// Mitsubishi GX Works2 project: elevator-finished-fixed   PLC: FX3U/FX3UC

PROGRAM MAIN
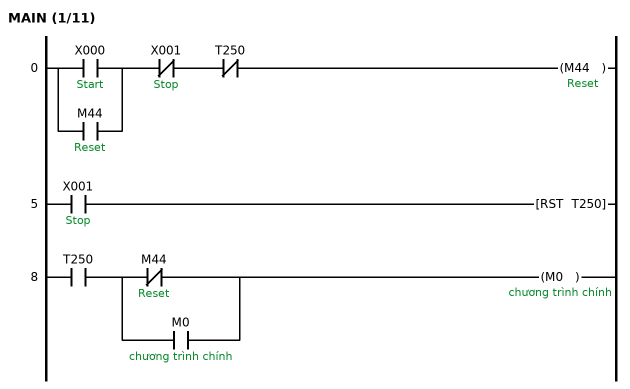
0     LD      X000  ; Start
      OR      M44  ; Reset
      ANI     X001  ; Stop
      ANI     T250
      OUT     M44  ; Reset
5     LD      X001  ; Stop
      RST     T250
8     LD      T250
      LDI     M44  ; Reset
      OR      M0  ; chương trình chính
      ANB
      OUT     M0  ; chương trình chính
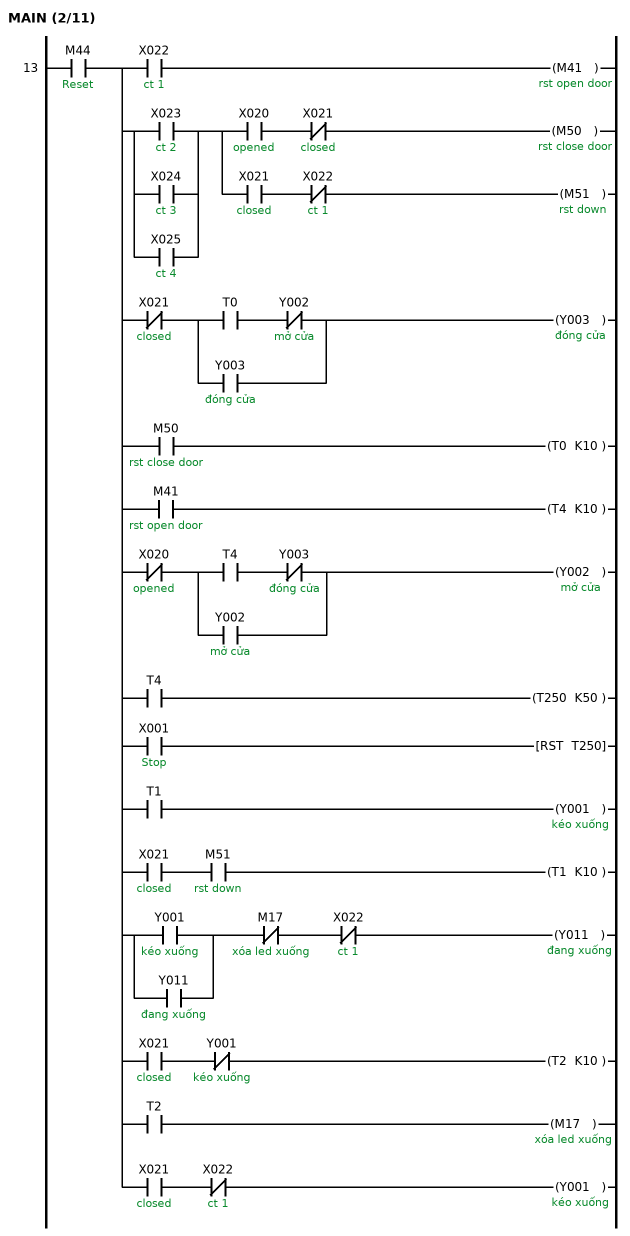
13    LD      M44  ; Reset
      MPS
      AND     X022  ; ct 1
      OUT     M41  ; rst open door
      MRD
      LD      X023  ; ct 2
      OR      X024  ; ct 3
      OR      X025  ; ct 4
      ANB
      MPS
      AND     X020  ; opened
      ANI     X021  ; closed
      OUT     M50  ; rst close door
      MPP
      AND     X021  ; closed
      ANI     X022  ; ct 1
      OUT     M51  ; rst down
      MRD
      ANI     X021  ; closed
      LD      T0
      ANI     Y002  ; mở cửa
      OR      Y003  ; đóng cửa
      ANB
      OUT     Y003  ; đóng cửa
      MRD
      AND     M50  ; rst close door
      OUT     T0 K10
      MRD
      AND     M41  ; rst open door
      OUT     T4 K10
      MRD
      ANI     X020  ; opened
      LD      T4
      ANI     Y003  ; đóng cửa
      OR      Y002  ; mở cửa
      ANB
      OUT     Y002  ; mở cửa
      MRD
      AND     T4
      OUT     T250 K50
      MRD
      AND     X001  ; Stop
      RST     T250
      MRD
      AND     T1
      OUT     Y001  ; kéo xuống
      MRD
      AND     X021  ; closed
      AND     M51  ; rst down
      OUT     T1 K10
      MRD
      LD      Y001  ; kéo xuống
      OR      Y011  ; đang xuống
      ANB
      ANI     M17  ; xóa led xuống
      ANI     X022  ; ct 1
      OUT     Y011  ; đang xuống
      MRD
      AND     X021  ; closed
      ANI     Y001  ; kéo xuống
      OUT     T2 K10
      MRD
      AND     T2
      OUT     M17  ; xóa led xuống
      MPP
      AND     X021  ; closed
      ANI     X022  ; ct 1
      OUT     Y001  ; kéo xuống
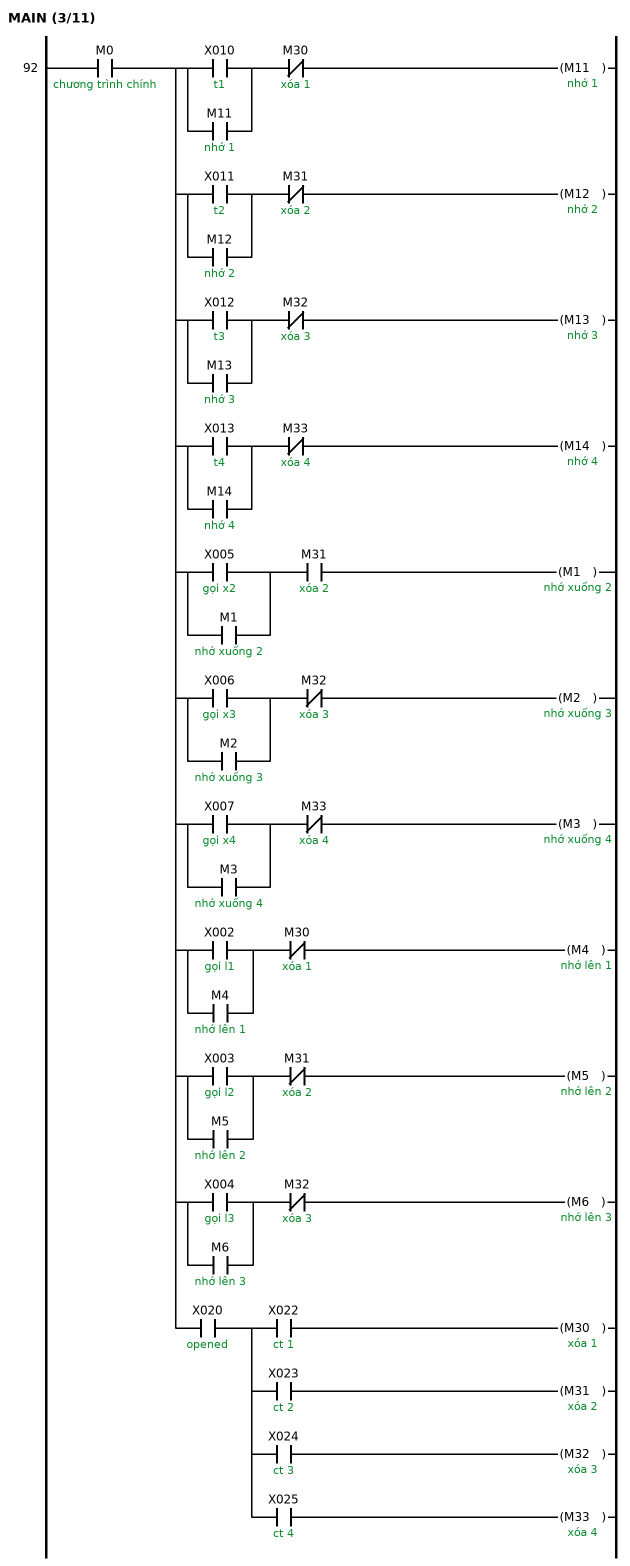
92    LD      M0  ; chương trình chính
      MPS
      LD      X010  ; t1
      OR      M11  ; nhớ 1
      ANB
      ANI     M30  ; xóa 1
      OUT     M11  ; nhớ 1
      MRD
      LD      X011  ; t2
      OR      M12  ; nhớ 2
      ANB
      ANI     M31  ; xóa 2
      OUT     M12  ; nhớ 2
      MRD
      LD      X012  ; t3
      OR      M13  ; nhớ 3
      ANB
      ANI     M32  ; xóa 3
      OUT     M13  ; nhớ 3
      MRD
      LD      X013  ; t4
      OR      M14  ; nhớ 4
      ANB
      ANI     M33  ; xóa 4
      OUT     M14  ; nhớ 4
      MRD
      LD      X005  ; gọi x2
      OR      M1  ; nhớ xuống 2
      ANB
      AND     M31  ; xóa 2
      OUT     M1  ; nhớ xuống 2
      MRD
      LD      X006  ; gọi x3
      OR      M2  ; nhớ xuống 3
      ANB
      ANI     M32  ; xóa 3
      OUT     M2  ; nhớ xuống 3
      MRD
      LD      X007  ; gọi x4
      OR      M3  ; nhớ xuống 4
      ANB
      ANI     M33  ; xóa 4
      OUT     M3  ; nhớ xuống 4
      MRD
      LD      X002  ; gọi l1
      OR      M4  ; nhớ lên 1
      ANB
      ANI     M30  ; xóa 1
      OUT     M4  ; nhớ lên 1
      MRD
      LD      X003  ; gọi l2
      OR      M5  ; nhớ lên 2
      ANB
      ANI     M31  ; xóa 2
      OUT     M5  ; nhớ lên 2
      MRD
      LD      X004  ; gọi l3
      OR      M6  ; nhớ lên 3
      ANB
      ANI     M32  ; xóa 3
      OUT     M6  ; nhớ lên 3
      MPP
      AND     X020  ; opened
      MPS
      AND     X022  ; ct 1
      OUT     M30  ; xóa 1
      MRD
      AND     X023  ; ct 2
      OUT     M31  ; xóa 2
      MRD
      AND     X024  ; ct 3
      OUT     M32  ; xóa 3
      MPP
      AND     X025  ; ct 4
      OUT     M33  ; xóa 4
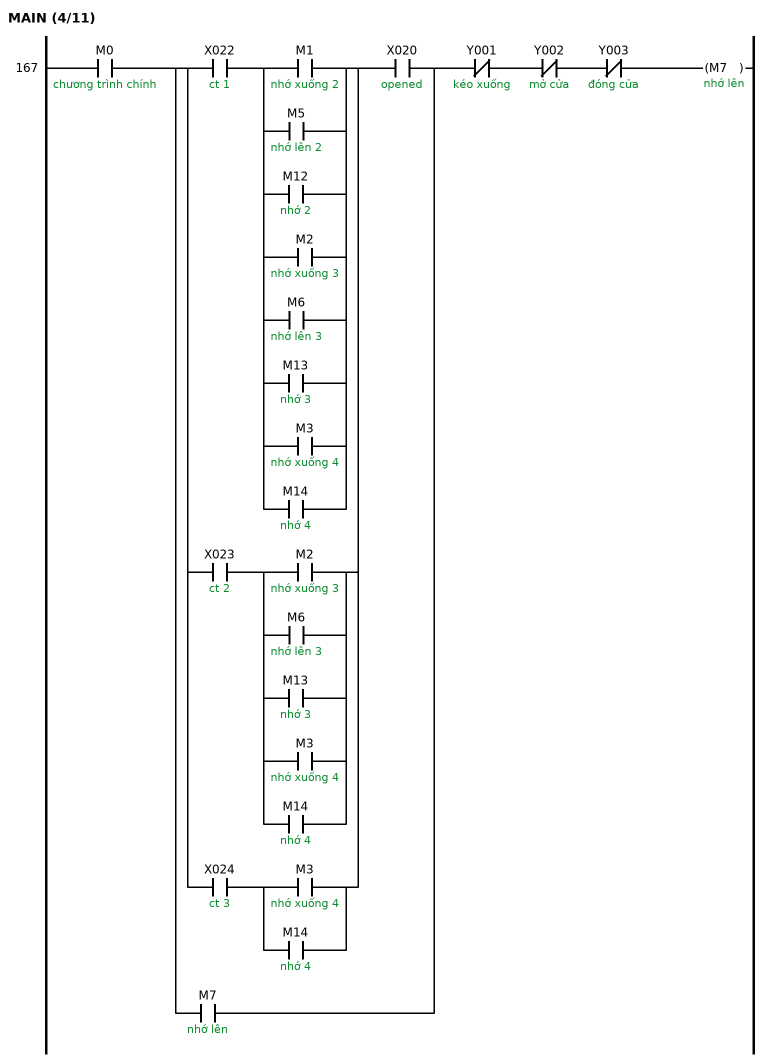
167   LD      M0  ; chương trình chính
      LD      X022  ; ct 1
      LD      M1  ; nhớ xuống 2
      OR      M5  ; nhớ lên 2
      OR      M12  ; nhớ 2
      OR      M2  ; nhớ xuống 3
      OR      M6  ; nhớ lên 3
      OR      M13  ; nhớ 3
      OR      M3  ; nhớ xuống 4
      OR      M14  ; nhớ 4
      ANB
      LD      X023  ; ct 2
      LD      M2  ; nhớ xuống 3
      OR      M6  ; nhớ lên 3
      OR      M13  ; nhớ 3
      OR      M3  ; nhớ xuống 4
      OR      M14  ; nhớ 4
      ANB
      ORB
      LD      X024  ; ct 3
      LD      M3  ; nhớ xuống 4
      OR      M14  ; nhớ 4
      ANB
      ORB
      AND     X020  ; opened
      OR      M7  ; nhớ lên
      ANB
      ANI     Y001  ; kéo xuống
      ANI     Y002  ; mở cửa
      ANI     Y003  ; đóng cửa
      OUT     M7  ; nhớ lên
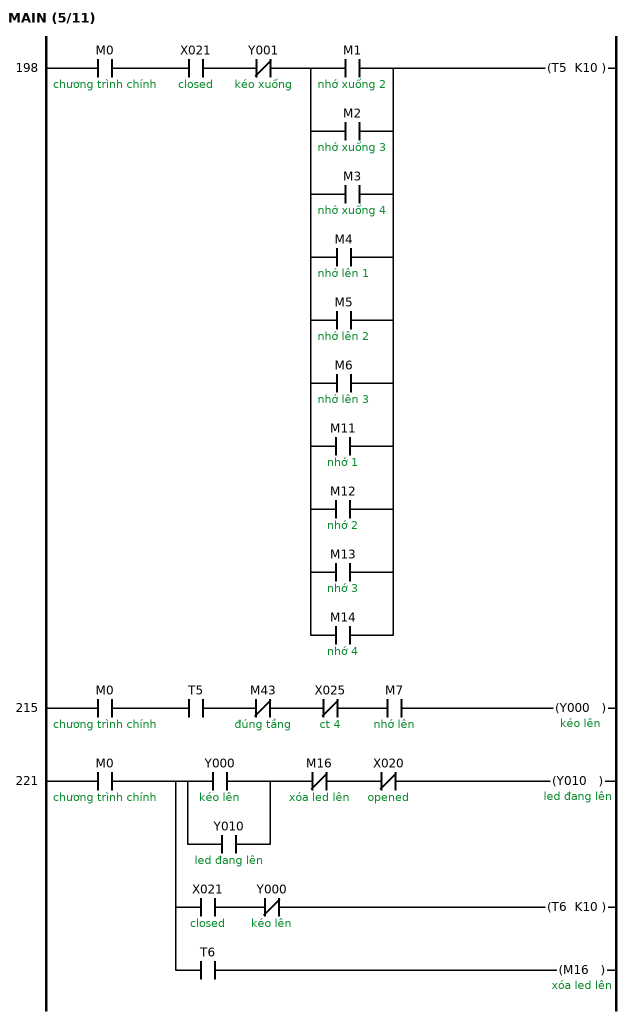
198   LD      M0  ; chương trình chính
      AND     X021  ; closed
      ANI     Y001  ; kéo xuống
      LD      M1  ; nhớ xuống 2
      OR      M2  ; nhớ xuống 3
      OR      M3  ; nhớ xuống 4
      OR      M4  ; nhớ lên 1
      OR      M5  ; nhớ lên 2
      OR      M6  ; nhớ lên 3
      OR      M11  ; nhớ 1
      OR      M12  ; nhớ 2
      OR      M13  ; nhớ 3
      OR      M14  ; nhớ 4
      ANB
      OUT     T5 K10
215   LD      M0  ; chương trình chính
      AND     T5
      ANI     M43  ; đúng tầng
      ANI     X025  ; ct 4
      AND     M7  ; nhớ lên
      OUT     Y000  ; kéo lên
221   LD      M0  ; chương trình chính
      MPS
      LD      Y000  ; kéo lên
      OR      Y010  ; led đang lên
      ANB
      ANI     M16  ; xóa led lên
      ANI     X020  ; opened
      OUT     Y010  ; led đang lên
      MRD
      AND     X021  ; closed
      ANI     Y000  ; kéo lên
      OUT     T6 K10
      MPP
      AND     T6
      OUT     M16  ; xóa led lên
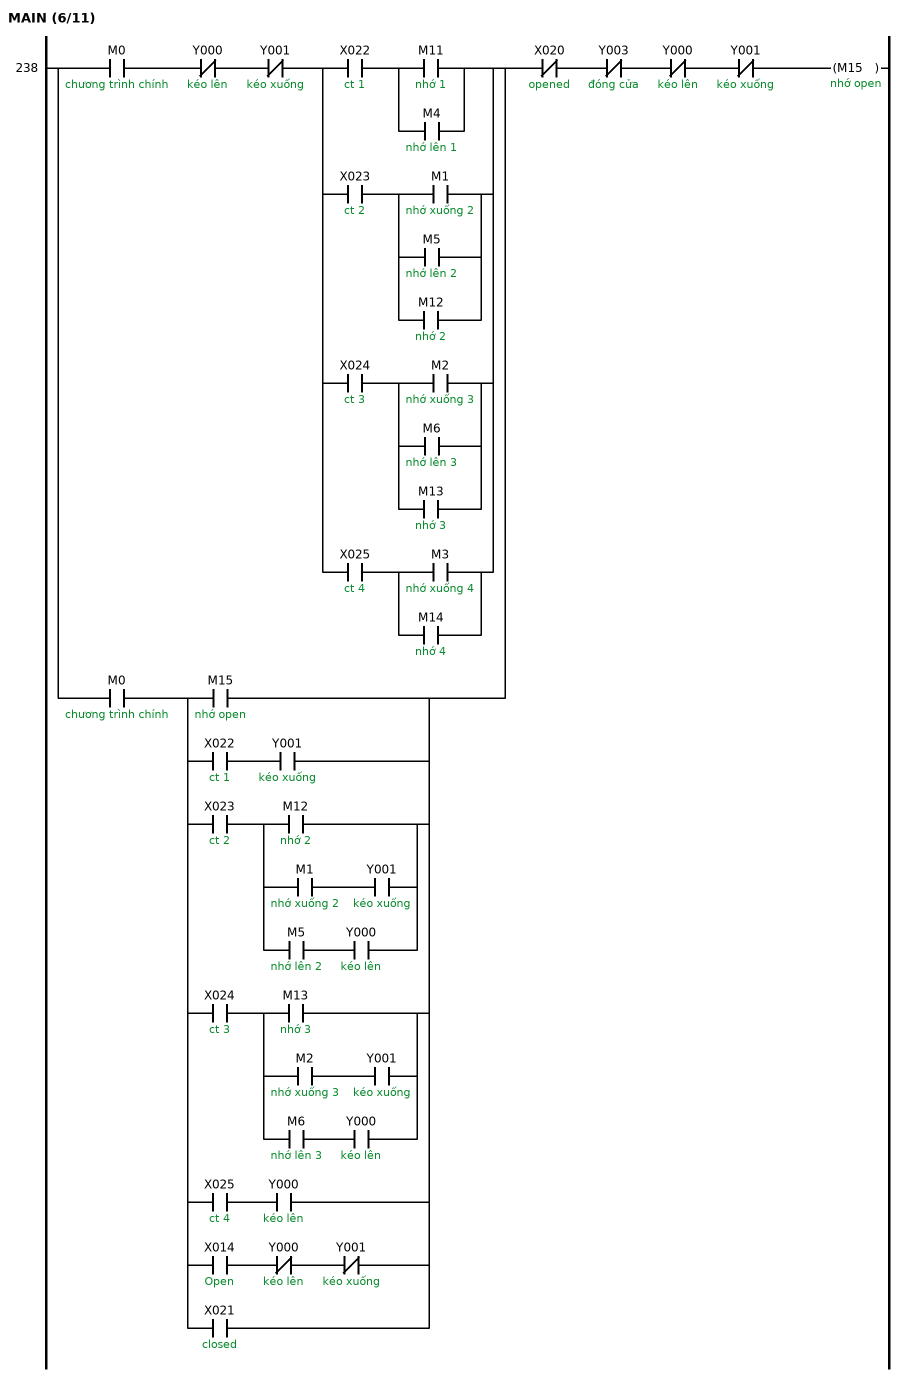
238   LD      M0  ; chương trình chính
      ANI     Y000  ; kéo lên
      ANI     Y001  ; kéo xuống
      LD      X022  ; ct 1
      LD      M11  ; nhớ 1
      OR      M4  ; nhớ lên 1
      ANB
      LD      X023  ; ct 2
      LD      M1  ; nhớ xuống 2
      OR      M5  ; nhớ lên 2
      OR      M12  ; nhớ 2
      ANB
      ORB
      LD      X024  ; ct 3
      LD      M2  ; nhớ xuống 3
      OR      M6  ; nhớ lên 3
      OR      M13  ; nhớ 3
      ANB
      ORB
      LD      X025  ; ct 4
      LD      M3  ; nhớ xuống 4
      OR      M14  ; nhớ 4
      ANB
      ORB
      ANB
      LD      M0  ; chương trình chính
      LD      M15  ; nhớ open
      LD      X022  ; ct 1
      AND     Y001  ; kéo xuống
      ORB
      LD      X023  ; ct 2
      LD      M12  ; nhớ 2
      LD      M1  ; nhớ xuống 2
      AND     Y001  ; kéo xuống
      ORB
      LD      M5  ; nhớ lên 2
      AND     Y000  ; kéo lên
      ORB
      ANB
      ORB
      LD      X024  ; ct 3
      LD      M13  ; nhớ 3
      LD      M2  ; nhớ xuống 3
      AND     Y001  ; kéo xuống
      ORB
      LD      M6  ; nhớ lên 3
      AND     Y000  ; kéo lên
      ORB
      ANB
      ORB
      LD      X025  ; ct 4
      AND     Y000  ; kéo lên
      ORB
      LD      X014  ; Open
      ANI     Y000  ; kéo lên
      ANI     Y001  ; kéo xuống
      ORB
      OR      X021  ; closed
      ANB
      ORB
      ANI     X020  ; opened
      ANI     Y003  ; đóng cửa
      ANI     Y000  ; kéo lên
      ANI     Y001  ; kéo xuống
      OUT     M15  ; nhớ open
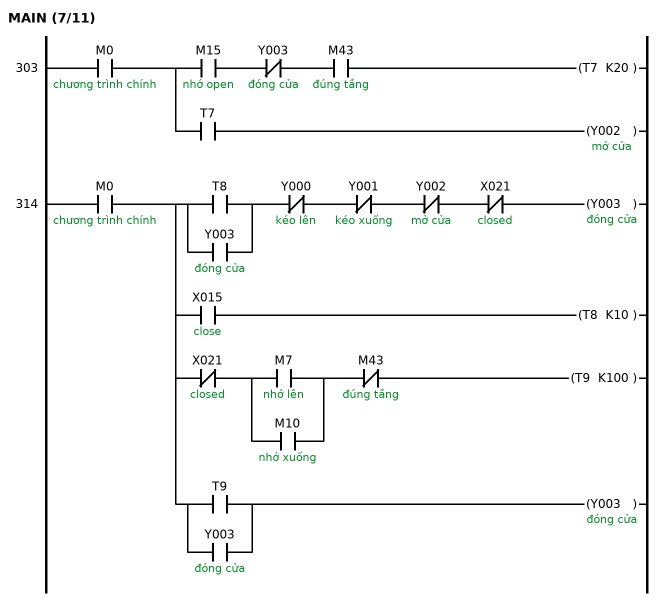
303   LD      M0  ; chương trình chính
      MPS
      AND     M15  ; nhớ open
      ANI     Y003  ; đóng cửa
      AND     M43  ; đúng tầng
      OUT     T7 K20
      MPP
      AND     T7
      OUT     Y002  ; mở cửa
314   LD      M0  ; chương trình chính
      MPS
      LD      T8
      OR      Y003  ; đóng cửa
      ANB
      ANI     Y000  ; kéo lên
      ANI     Y001  ; kéo xuống
      ANI     Y002  ; mở cửa
      ANI     X021  ; closed
      OUT     Y003  ; đóng cửa
      MRD
      AND     X015  ; close
      OUT     T8 K10
      MRD
      ANI     X021  ; closed
      LD      M7  ; nhớ lên
      OR      M10  ; nhớ xuống
      ANB
      ANI     M43  ; đúng tầng
      OUT     T9 K100
      MPP
      LD      T9
      OR      Y003  ; đóng cửa
      ANB
      OUT     Y003  ; đóng cửa
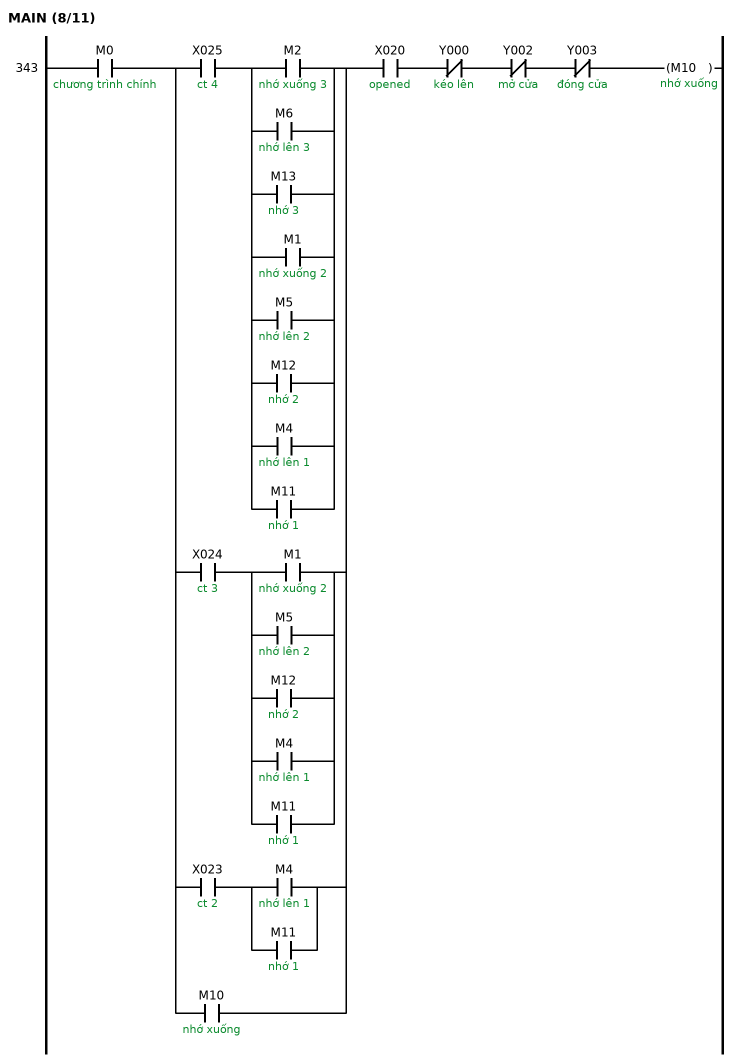
343   LD      M0  ; chương trình chính
      LD      X025  ; ct 4
      LD      M2  ; nhớ xuống 3
      OR      M6  ; nhớ lên 3
      OR      M13  ; nhớ 3
      OR      M1  ; nhớ xuống 2
      OR      M5  ; nhớ lên 2
      OR      M12  ; nhớ 2
      OR      M4  ; nhớ lên 1
      OR      M11  ; nhớ 1
      ANB
      LD      X024  ; ct 3
      LD      M1  ; nhớ xuống 2
      OR      M5  ; nhớ lên 2
      OR      M12  ; nhớ 2
      OR      M4  ; nhớ lên 1
      OR      M11  ; nhớ 1
      ANB
      ORB
      LD      X023  ; ct 2
      LD      M4  ; nhớ lên 1
      OR      M11  ; nhớ 1
      ANB
      ORB
      OR      M10  ; nhớ xuống
      ANB
      AND     X020  ; opened
      ANI     Y000  ; kéo lên
      ANI     Y002  ; mở cửa
      ANI     Y003  ; đóng cửa
      OUT     M10  ; nhớ xuống
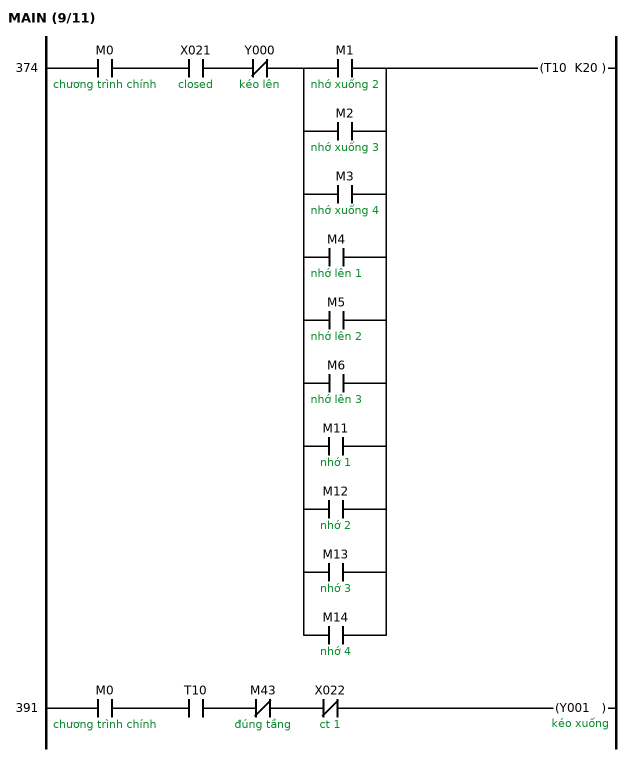
374   LD      M0  ; chương trình chính
      AND     X021  ; closed
      ANI     Y000  ; kéo lên
      LD      M1  ; nhớ xuống 2
      OR      M2  ; nhớ xuống 3
      OR      M3  ; nhớ xuống 4
      OR      M4  ; nhớ lên 1
      OR      M5  ; nhớ lên 2
      OR      M6  ; nhớ lên 3
      OR      M11  ; nhớ 1
      OR      M12  ; nhớ 2
      OR      M13  ; nhớ 3
      OR      M14  ; nhớ 4
      ANB
      OUT     T10 K20
391   LD      M0  ; chương trình chính
      AND     T10
      ANI     M43  ; đúng tầng
      ANI     X022  ; ct 1
      OUT     Y001  ; kéo xuống
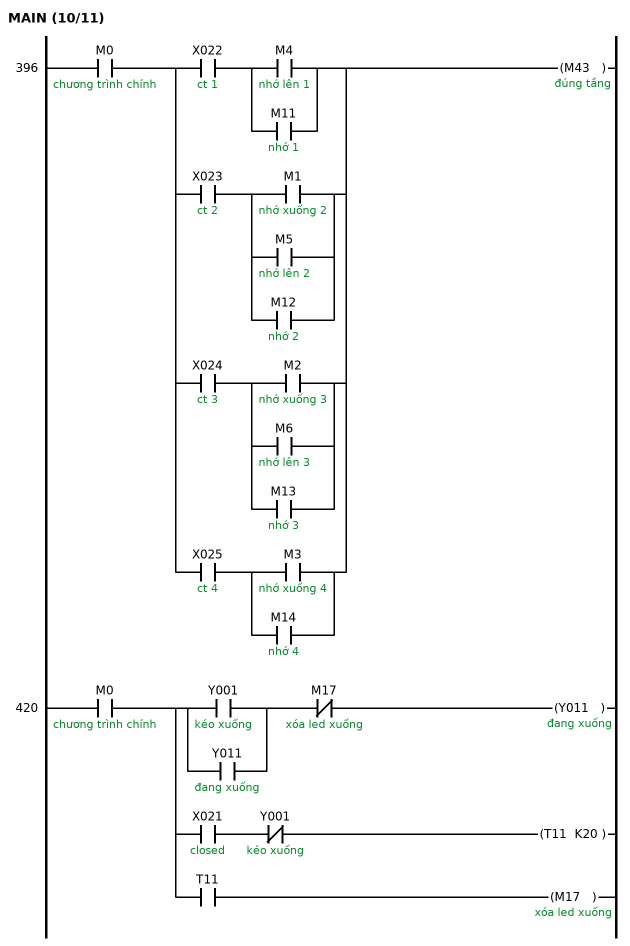
396   LD      M0  ; chương trình chính
      LD      X022  ; ct 1
      LD      M4  ; nhớ lên 1
      OR      M11  ; nhớ 1
      ANB
      LD      X023  ; ct 2
      LD      M1  ; nhớ xuống 2
      OR      M5  ; nhớ lên 2
      OR      M12  ; nhớ 2
      ANB
      ORB
      LD      X024  ; ct 3
      LD      M2  ; nhớ xuống 3
      OR      M6  ; nhớ lên 3
      OR      M13  ; nhớ 3
      ANB
      ORB
      LD      X025  ; ct 4
      LD      M3  ; nhớ xuống 4
      OR      M14  ; nhớ 4
      ANB
      ORB
      ANB
      OUT     M43  ; đúng tầng
420   LD      M0  ; chương trình chính
      MPS
      LD      Y001  ; kéo xuống
      OR      Y011  ; đang xuống
      ANB
      ANI     M17  ; xóa led xuống
      OUT     Y011  ; đang xuống
      MRD
      AND     X021  ; closed
      ANI     Y001  ; kéo xuống
      OUT     T11 K20
      MPP
      AND     T11
      OUT     M17  ; xóa led xuống
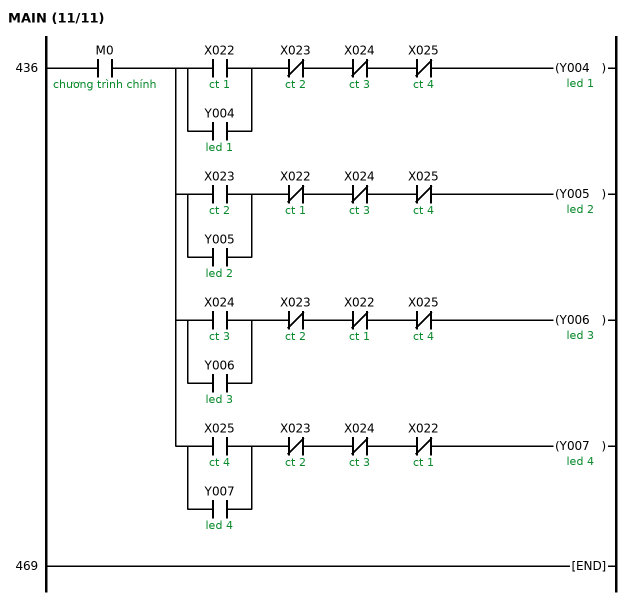
436   LD      M0  ; chương trình chính
      MPS
      LD      X022  ; ct 1
      OR      Y004  ; led 1
      ANB
      ANI     X023  ; ct 2
      ANI     X024  ; ct 3
      ANI     X025  ; ct 4
      OUT     Y004  ; led 1
      MRD
      LD      X023  ; ct 2
      OR      Y005  ; led 2
      ANB
      ANI     X022  ; ct 1
      ANI     X024  ; ct 3
      ANI     X025  ; ct 4
      OUT     Y005  ; led 2
      MRD
      LD      X024  ; ct 3
      OR      Y006  ; led 3
      ANB
      ANI     X023  ; ct 2
      ANI     X022  ; ct 1
      ANI     X025  ; ct 4
      OUT     Y006  ; led 3
      MPP
      LD      X025  ; ct 4
      OR      Y007  ; led 4
      ANB
      ANI     X023  ; ct 2
      ANI     X024  ; ct 3
      ANI     X022  ; ct 1
      OUT     Y007  ; led 4
469   END
END_PROGRAM
